// TIA Portal V16 export
// export: Created 2024-09-05T17:39:10.3491384Z, ExportSetting WithDefaults, DisplayName Totally Integrated Automation Portal, DisplayVersion V16 Update 6, DisplayName TIA Portal Version Control Interface, DisplayVersion V16 Update 2, DisplayName TIA Portal Openness, DisplayVersion V16 Update 6, DisplayName STEP 7 Professional, DisplayVersion V16 Update 6, DisplayName STEP 7 Safety, DisplayVersion V16, DisplayName WinCC Advanced, DisplayVersion V16 Update 6
FUNCTION_BLOCK "HydraulicMotor"   // FB36, LAD
{ S7_Optimized_Access := 'TRUE' }
VERSION : 0.1
// stored: AutoNumber true, IsIECCheckEnabled false, IsRetainMemResEnabled false, MemoryReserve 100, SetENOAutomatically false, UDAEnableTagReadback false
   VAR_INPUT
      cycleActiveCupforming : Bool;
      cycleActiveRiveting : Bool;
      temp1nok : Bool;
      temp2nok : Bool;
   END_VAR
   VAR_IN_OUT
      data : "UDT_HydraulicPump";
      qKM20 : Bool;
      qMotor : Bool;
      qValveCupforming : Bool;
      qValveRiveting : Bool;
   END_VAR
   VAR
      R_TRIG_Instance { S7_SetPoint := 'True'} : R_TRIG;
      cnt { S7_SetPoint := 'True'} : Int;
      IEC_Timer_0_Instance { S7_SetPoint := 'True'} : TON_TIME;
      F_TRIG_Instance { S7_SetPoint := 'True'} : F_TRIG;
      IEC_Timer_0_Instance_1 { S7_SetPoint := 'True'} : TON_TIME;
   END_VAR
   VAR_TEMP   // added for the SCL form of the ladder/FBD networks
      _w1 : Bool;
   END_VAR
BEGIN

REGION Network 1: Start auto mode
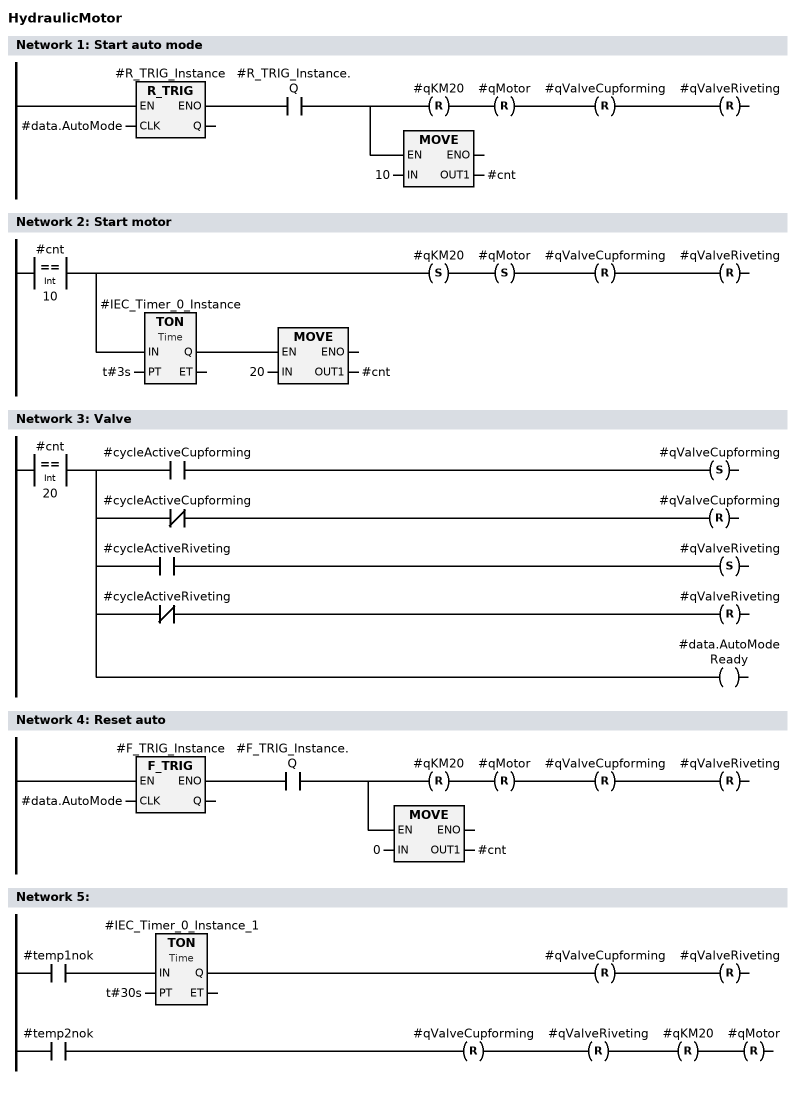
   RUNG wire#powerrail
      #R_TRIG_Instance.R_TRIG(CLK := #data.AutoMode, Q =>)
      Contact( #R_TRIG_Instance.Q )
      wire#w1
      R_Coil( #qKM20 )
      R_Coil( #qMotor )
      R_Coil( #qValveCupforming )
      R_Coil( #qValveRiveting )
   END_RUNG
   RUNG wire#w1
      Move(in := 10, out1 => #cnt)
   END_RUNG
   // the same network as SCL:
   #R_TRIG_Instance(CLK := #data.AutoMode, ENO => #_w1);   // R_TRIG
   IF #_w1 AND #R_TRIG_Instance.Q THEN
       #qKM20 := FALSE;
       #qMotor := FALSE;
       #qValveCupforming := FALSE;
       #qValveRiveting := FALSE;
       #cnt := 10;
   END_IF;
END_REGION

REGION Network 2: Start motor
   RUNG wire#powerrail
      { S7_Templates := "SrcType := Int" } EQ_Contact(in1 := #cnt, in2 := 10)
      wire#w1
      S_Coil( #qKM20 )
      S_Coil( #qMotor )
      R_Coil( #qValveCupforming )
      R_Coil( #qValveRiveting )
   END_RUNG
   RUNG wire#w1
      { S7_Templates := "time_type := Time" } #IEC_Timer_0_Instance.TON(pt := t#3s, et =>)
      Move(in := 20, out1 => #cnt)
   END_RUNG
   // the same network as SCL:
   #_w1 := #cnt = 10;
   IF #_w1 THEN
       #qKM20 := TRUE;
       #qMotor := TRUE;
       #qValveCupforming := FALSE;
       #qValveRiveting := FALSE;
   END_IF;
   #IEC_Timer_0_Instance(IN := #_w1, PT := t#3s);   // TON
   IF #IEC_Timer_0_Instance.Q THEN #cnt := 20; END_IF;
END_REGION

REGION Network 3: Valve
   RUNG wire#powerrail
      { S7_Templates := "SrcType := Int" } EQ_Contact(in1 := #cnt, in2 := 20)
      wire#w1
      Contact( #cycleActiveCupforming )
      S_Coil( #qValveCupforming )
   END_RUNG
   RUNG wire#w1
      I_Contact( #cycleActiveCupforming )
      R_Coil( #qValveCupforming )
   END_RUNG
   RUNG wire#w1
      Contact( #cycleActiveRiveting )
      S_Coil( #qValveRiveting )
   END_RUNG
   RUNG wire#w1
      I_Contact( #cycleActiveRiveting )
      R_Coil( #qValveRiveting )
   END_RUNG
   RUNG wire#w1
      Coil( #data.AutoModeReady )
   END_RUNG
   // the same network as SCL:
   #_w1 := #cnt = 20;
   IF #_w1 AND #cycleActiveCupforming THEN #qValveCupforming := TRUE; END_IF;
   IF #_w1 AND NOT #cycleActiveCupforming THEN #qValveCupforming := FALSE; END_IF;
   IF #_w1 AND #cycleActiveRiveting THEN #qValveRiveting := TRUE; END_IF;
   IF #_w1 AND NOT #cycleActiveRiveting THEN #qValveRiveting := FALSE; END_IF;
   #data.AutoModeReady := #_w1;
END_REGION

REGION Network 4: Reset auto
   RUNG wire#powerrail
      #F_TRIG_Instance.F_TRIG(CLK := #data.AutoMode, Q =>)
      Contact( #F_TRIG_Instance.Q )
      wire#w1
      R_Coil( #qKM20 )
      R_Coil( #qMotor )
      R_Coil( #qValveCupforming )
      R_Coil( #qValveRiveting )
   END_RUNG
   RUNG wire#w1
      Move(in := 0, out1 => #cnt)
   END_RUNG
   // the same network as SCL:
   #F_TRIG_Instance(CLK := #data.AutoMode, ENO => #_w1);   // F_TRIG
   IF #_w1 AND #F_TRIG_Instance.Q THEN
       #qKM20 := FALSE;
       #qMotor := FALSE;
       #qValveCupforming := FALSE;
       #qValveRiveting := FALSE;
       #cnt := 0;
   END_IF;
END_REGION

REGION Network 5
   RUNG wire#powerrail
      Contact( #temp1nok )
      { S7_Templates := "time_type := Time" } #IEC_Timer_0_Instance_1.TON(pt := t#30s, et =>)
      R_Coil( #qValveCupforming )
      R_Coil( #qValveRiveting )
   END_RUNG
   RUNG wire#powerrail
      Contact( #temp2nok )
      R_Coil( #qValveCupforming )
      R_Coil( #qValveRiveting )
      R_Coil( #qKM20 )
      R_Coil( #qMotor )
   END_RUNG
   // the same network as SCL:
   #IEC_Timer_0_Instance_1(IN := #temp1nok, PT := t#30s);   // TON
   IF #IEC_Timer_0_Instance_1.Q THEN
       #qValveCupforming := FALSE;
       #qValveRiveting := FALSE;
   END_IF;
   IF #temp2nok THEN
       #qValveCupforming := FALSE;
       #qValveRiveting := FALSE;
       #qKM20 := FALSE;
       #qMotor := FALSE;
   END_IF;
END_REGION
END_FUNCTION_BLOCK
